(* IEC 61131-3 sources: PLC_problems-ladder-diagram-/problem(5)/build, 2 files *)

(* ---- plc.st ---- *)
TYPE
  LOGLEVEL : (CRITICAL, WARNING, INFO, DEBUG) := INFO;
END_TYPE

FUNCTION_BLOCK LOGGER
  VAR_INPUT
    TRIG : BOOL;
    MSG : STRING;
    LEVEL : LOGLEVEL := INFO;
  END_VAR
  VAR
    TRIG0 : BOOL;
  END_VAR

  IF TRIG AND NOT TRIG0 THEN
  {{
   LogMessage(GetFbVar(LEVEL),(char*)GetFbVar(MSG, .body),GetFbVar(MSG, .len));
  }}
  END_IF;
  TRIG0:=TRIG;
END_FUNCTION_BLOCK

PROGRAM program0
  VAR
    staff1 : BOOL;
    staff2 : BOOL;
    bio1 : BOOL;
    bio2 : BOOL;
    bio3 : BOOL;
    HEAD : BOOL;
    DOOR_OPEN : BOOL;
  END_VAR

  DOOR_OPEN := HEAD OR (bio2 AND bio1 OR bio3 AND bio1 OR bio3 AND bio2) AND staff2 AND staff1;
END_PROGRAM

CONFIGURATION Config0

  RESOURCE Res0 ON PLC
    TASK task0(INTERVAL := T#20ms,PRIORITY := 0);
    PROGRAM instance0 WITH task0 : program0;
  END_RESOURCE
END_CONFIGURATION

(* ---- generated_plc.st ---- *)
PROGRAM program0
  VAR
    staff1 : BOOL;
    staff2 : BOOL;
    bio1 : BOOL;
    bio2 : BOOL;
    bio3 : BOOL;
    HEAD : BOOL;
    DOOR_OPEN : BOOL;
  END_VAR

  DOOR_OPEN := HEAD OR (bio2 AND bio1 OR bio3 AND bio1 OR bio3 AND bio2) AND staff2 AND staff1;
END_PROGRAM

CONFIGURATION Config0

  RESOURCE Res0 ON PLC
    TASK task0(INTERVAL := T#20ms,PRIORITY := 0);
    PROGRAM instance0 WITH task0 : program0;
  END_RESOURCE
END_CONFIGURATION
